{attribute 'qualified_only'}
VAR_GLOBAL	
	B1  AT %I* :BOOL; 	// Lichtschranke 0°
	B2  AT %I* :BOOL;   // Lichtschranke 45° CCW
	S1  AT %I*:BOOL;   // Taster (①) → Schliesser
	S2  AT %I*:BOOL;   // Taster (⓪) → Öffner
	S3  AT %I*:BOOL;   // Taster (Ⅰ) → Schliesser
	S4  AT %I*:BOOL;   // Taster (STOP) → Öffner
	S5  AT %I*:BOOL;   // Taster (Ⅱ) → Schliesser
	S6  AT %I*:BOOL;   // Taster (←) → Schliesser
	S7  AT %I* :BOOL;   // Taster (STOP) → Öffner
	S8  AT %I*:BOOL;   // Taster (→) → Schliesser
	S91 AT %I*:BOOL;   // Not-Halt → Schliesser
	S92 AT %I*:BOOL;   // Not-Halt → Öffner	
END_VAR

(* stored: Version 1.1.0.1, ProductVersion 3.1.4024.5
   GVL DI: Id {c2d05302-d374-4f85-80dd-41006a3e3277} *)
